{attribute 'qualified_only'}
{attribute 'strict'}
TYPE SystemStatesRunMode :
(
	Off := 0, LowSpeed, HighSpeed
);
END_TYPE

(* stored: Version 1.1.0.1, ProductVersion 3.1.4024.6
   DUT SystemStatesRunMode: Id {8e5b585e-9d16-4661-b044-0658e4f58697} *)
